Fanuc KAREL source: kt00039.KL

-- PROVISIONAL review KL for V770-1; original PC SHA256 f4571f5d26b74029cf2620b801130812c5ff7c7cee1044c7028a0ca49c6bc60b
-- Incomplete behavior may be omitted. Consult companion uncertainty JSON. Do not deploy.
PROGRAM KT00039
%NOLOCKGROUP
VAR
  I1 : INTEGER
  OUT : INTEGER
-- UNRESOLVED_DECL H2 type=002017
BEGIN
  -- UNRESOLVED_PC offsets 5-16; opcodes 2E,23
  -- UNRESOLVED_PC offsets 21-35; opcodes 2E,22,9D,33,B4
  -- UNRESOLVED_PC offsets 40-62; opcodes 21,22,9D,33,B3,53,23
  -- UNRESOLVED_PC offsets 67-71; opcodes 7F
END KT00039
